{attribute 'GeneratedUsingTerminal: CU1128--0000'}
{attribute addProperty BoxType "CU1128--0000"}
{attribute addProperty Id "InfoDataAT %I*InfoData_6F19DB2B2"}
{attribute addProperty CRC "532711307"}
{attribute addProperty Size "2"}
TYPE CU1128_1FC0878B EXTENDS EtcSlaveTerminalBase_947E5A46 :
STRUCT
	{attribute addProperty Name "InfoData"}
	InfoData : InfoData_6F19DB2B;
END_STRUCT
END_TYPE

(* stored: Version 1.2.0.0, ProductVersion 3.1.4024.9
   DUT CU1128_1FC0878B: Id {deca1447-8be5-49a1-9b1f-fa28f4f618db} *)
